FUNCTION_BLOCK FB_LUTDevice EXTENDS FD_Device 
VAR_INPUT
END_VAR

VAR_OUTPUT
END_VAR

VAR
	//===================== Variable
	eLTUPosition					: E_LTUPosition;
	bCarrierPresent				: BOOL;
	bLTUFree							: BOOL;
	
	bReserved							: BOOL;
	eReservedBy						: E_Convoyer;
	
	
	
	//===================== Instance
	fbPneuCyl3Pos_AxisZ								: FB_PneuCyl_3Pos     	 (GVL_Customer.C_Name_LTUPneuClyZ,
																															GVL_Customer.C_ID_LTUPneuClyZ
																										  				); 
																													
	fbStopperLut											: FB_PneuCyl_Stopper     (GVL_Customer.C_Name_LUTStopper,
																															GVL_Customer.C_ID_LUTStopper
																										  			 );																												
																													
	fbLUTLightBarrier									: FB_Input					  		(GVL_Customer.C_Name_LUTLightBarrier,
																															GVL_Customer.C_ID_LUTLightBarrier
																										  				);																																										
	
	fbLUTSimpleMotor									: FB_SimpleMotor      		(GVL_Customer.C_Name_LUTDcMotor,
																															GVL_Customer.C_ID_LUTSimpleMotor
																										  				);

																										
END_VAR

VAR CONSTANT
	// --------------------------Base------------------
	C_SeqStep_OnBasePos_Start								: UINT :=  20; 
	C_SeqStep_OnBasePos_WaitOpMode					: UINT :=  30;
	C_SeqStep_OnBasePos_Done								: UINT :=  100; 
	
	// --------------------------Auto Sequence------------------
	
	C_SeqStep_Auto_Start										: UINT :=  200;
	C_SeqStep_Auto_End											: UINT :=  400;
END_VAR


//******* Important and necessary
SUPER^();  
//====================================
IF NOT Enable THEN RETURN; END_IF

fbPneuCyl3Pos_AxisZ();
fbStopperLut();
fbLUTLightBarrier();
fbLUTSimpleMotor();

PROPERTY CarrierPresent : BOOL
GET
CarrierPresent := bCarrierPresent;
END_GET
SET
bCarrierPresent := CarrierPresent;
END_SET
END_PROPERTY

//FB_Init ist immer implizit verfügbar und wird primär für die Initialisierung verwendet.
//Der Rückgabewert wird nicht ausgewertet. Für gezielte Einflussnahme können Sie
//die Methoden explizit deklarieren und darin mit dem Standard-Initialisierungscode 
//zusätzlichen Code bereitstellen. Sie können den Rückgabewert auswerten.
METHOD FB_Init: BOOL
VAR_INPUT    
	bInitRetains					: BOOL; 					// TRUE: Die Retain-Variablen werden initialisiert (Reset warm / Reset kalt)    
	bInCopyCode						: BOOL;  					// TRUE: Die Instanz wird danach in den Kopiercode kopiert (Online-Change)
	
	I_Name                : STRING;         //  Name
	I_ID                  : UINT;           // ID
  I_itfOwner					  : ITF_Owner;      // owner 
END_VAR
END_METHOD

PROPERTY LTUFree : BOOL
GET

LTUFree := bLTUFree;
END_GET
SET
bLTUFree := LTUFree;
END_SET
END_PROPERTY

PROPERTY LTUPosition : E_LTUPosition
GET
LTUPosition := eLTUPosition;
END_GET
SET
eLTUPosition := LTUPosition;
END_SET
END_PROPERTY

METHOD mAutomatic : E_CmdState
VAR_INPUT
	I_bExecute	: BOOL;
END_VAR
END_METHOD

METHOD mCmdExec_Auto : E_CmdState
VAR_INPUT
END_VAR

CASE SequenceID OF

  //******************************************************* Idle 
  C_SeqStep_Idle: 
  	SequenceID       :=  C_SeqStep_Start;
  
  //****************************************************** Start
  C_SeqStep_Start:
  	
  	SequenceID       :=  C_SeqStep_OnBasePos_Start;
	C_SeqStep_OnBasePos_Start:
	
		SequenceID       :=  C_SeqStep_Done;;
	
//	C_SeqStep_OnBasePos_Start:
	
	
//	C_SeqStep_OnBasePos_Start:
	
	
  C_SeqStep_Error: 
    //************* all FB reset

		//************* 
    mCmdExec_Auto := mDone(); 
  //**********************Done 
  	
 	C_SeqStep_Done:
  	mCmdExec_Auto := mDone();

END_CASE
END_METHOD

METHOD mCmdExec_Homing : E_CmdState
VAR_INPUT
END_VAR

CASE SequenceID OF

  //******************************************************* Idle 
  C_SeqStep_Idle: 
  	SequenceID       :=  C_SeqStep_Start;
  
  //****************************************************** Start
  C_SeqStep_Start:
   
  	SequenceID       :=  C_SeqStep_Done;
	
  C_SeqStep_Error: 
    //************* all FB reset

		//************* 
    mCmdExec_Homing := mDone(); 
  //**********************Done 
 
 	C_SeqStep_Done:
  	mCmdExec_Homing := mDone();

END_CASE
END_METHOD

METHOD mCmdExec_MoveBottom : E_CmdState
VAR_INPUT
	I_bExecute					: BOOL;
END_VAR

VAR
	L_eCmdState 					: E_CmdState;
END_VAR
// No command requested.
IF NOT I_bExecute 
	THEN
  	mCmdExec_MoveMiddle := E_CmdState.Idle;
    RETURN;
END_IF

// Move vertical axis to TOP.
L_eCmdState := fbPneuCyl3Pos_AxisZ.mCallBottom(TRUE);
CASE L_eCmdState OF
	E_CmdState.Succeeded:
  	mCmdExec_MoveBottom := E_CmdState.Succeeded;
  E_CmdState.Busy:
  	mCmdExec_MoveBottom := E_CmdState.Busy;
ELSE
	mCmdExec_MoveBottom := L_eCmdState;
END_CASE
END_METHOD

METHOD mCmdExec_MoveMiddle : E_CmdState
VAR_INPUT
	I_bExecute					: BOOL;
END_VAR

VAR
	L_eCmdState 					: E_CmdState;
END_VAR
// No command requested.
IF NOT I_bExecute 
	THEN
  	mCmdExec_MoveMiddle := E_CmdState.Idle;
    RETURN;
END_IF

// Move vertical axis to TOP.
L_eCmdState := fbPneuCyl3Pos_AxisZ.mCallMiddle(TRUE);
CASE L_eCmdState OF
	E_CmdState.Succeeded:
  	mCmdExec_MoveMiddle := E_CmdState.Succeeded;
  E_CmdState.Busy:
  	mCmdExec_MoveMiddle := E_CmdState.Busy;
ELSE
	mCmdExec_MoveMiddle := L_eCmdState;
END_CASE
END_METHOD

METHOD mCmdExec_MoveTop : E_CmdState
VAR_INPUT
	I_bExecute					: BOOL;
END_VAR

VAR
	L_eCmdState 					: E_CmdState;
END_VAR
// No command requested.
IF NOT I_bExecute 
	THEN
  	mCmdExec_MoveTop := E_CmdState.Idle;
    RETURN;
END_IF

// Move vertical axis to TOP.
L_eCmdState := fbPneuCyl3Pos_AxisZ.mCallTop(TRUE);
CASE L_eCmdState OF
	E_CmdState.Succeeded:
  	mCmdExec_MoveTop := E_CmdState.Succeeded;
  E_CmdState.Busy:
  	mCmdExec_MoveTop := E_CmdState.Busy;
ELSE
	mCmdExec_MoveTop := L_eCmdState;
END_CASE
END_METHOD

METHOD mCmdExec_Service : E_CmdState
VAR_INPUT
END_VAR
;
END_METHOD

METHOD mCmdExec_TransferTop : E_CmdState
VAR_INPUT
	I_bExecute					: BOOL;
END_VAR
// No command requested.
IF NOT I_bExecute THEN
    fbLUTSimpleMotor.mStopMotor(TRUE);
    mCmdExec_TransferTop := E_CmdState.Idle;
    RETURN;
END_IF

// Start LTU motor for top transfer.
fbLUTSimpleMotor.mStartMotor(TRUE);

// Wait  carrier leaves LTU.
IF NOT fbStopperLut.CarriePresent 
	THEN
    fbLUTSimpleMotor.mStopMotor(TRUE);
    mCmdExec_TransferTop := E_CmdState.Succeeded;
    RETURN;
END_IF

mCmdExec_TransferTop := E_CmdState.Busy;
END_METHOD

METHOD mHold : E_CmdState
VAR_INPUT
	I_bExecute	: BOOL;
END_VAR

SUPER^.mHold(I_bExecute);
END_METHOD

METHOD mHome : E_CmdState
VAR_INPUT
	I_bExecute	: BOOL;
END_VAR

SUPER^.mHome(I_bExecute);
END_METHOD

METHOD mRelease : E_CmdState
VAR_INPUT
	I_bExecute	: BOOL;
END_VAR

SUPER^.mRelease(I_bExecute);
END_METHOD

METHOD mSequence : E_CmdState
VAR_INPUT
	I_bExecute				: BOOL;
END_VAR

VAR
	L_eState 					: E_CmdState;
END_VAR
mSequence := SUPER^.mSequence(I_bExecute);	


// Generic checks from parent
L_eState := SUPER^.mSequence(I_bExecute := I_bExecute);

IF L_eState <> E_CmdState.Busy 
	THEN
    mSequence := L_eState;
    RETURN;
END_IF

CASE Mode OF
	E_Mode.Homing:
		mSequence := mCmdExec_Homing();
		
	E_Mode.Auto:
		mSequence := mCmdExec_Auto();
		
	E_Mode.Service:
		mSequence := mCmdExec_Service();
		
END_CASE
END_METHOD

METHOD mService : E_CmdState
VAR_INPUT
	I_bExecute	: BOOL;
END_VAR

SUPER^.mService(I_bExecute);
END_METHOD

METHOD mStop : E_CmdState
VAR_INPUT
	I_bExecute	: BOOL;
END_VAR

SUPER^.mStop(I_bExecute);
END_METHOD

PROPERTY ReservedBy : E_Convoyer
GET
ReservedBy := eReservedBy;
END_GET
SET
eReservedBy := ReservedBy;
END_SET
END_PROPERTY

END_FUNCTION_BLOCK

(* stored: Version 1.1.0.1, ProductVersion 3.1.4026.18
   POU FB_LUTDevice: Id {1d37f6f4-ced3-4fc7-b8fb-537fe5b0ee0b}, SpecialFunc None
   Folder 01 Properties: Id {01153c84-2cbf-4774-9afe-06465af82a17}
   Folder 02 Methodes: Id {1154e57b-5607-4e8c-9894-d39905ffa9c5}
   Folder 100 CmdExecute: Id {737ecdee-bdd3-4011-be43-9c8053143eb0}
   Property CarrierPresent: Id {b074603b-40b1-4657-ab62-b1cd6acb861f}
   Get Get: Id {88207567-04e5-4568-82f0-781cf9a61ad4}
   Set Set: Id {fd122f58-f442-4621-8637-9e667fca0acd}
   Method FB_Init: Id {4e8aa732-d3ac-4d90-bbea-84986dfc142d}
   Property LTUFree: Id {1f84a690-a1f2-456d-ad2b-bc5117437904}
   Get Get: Id {d00d9a6b-7aca-4015-aa9d-f54e3711617d}
   Set Set: Id {d538fb44-3dfc-4c3c-8b31-3a15c25ffd6c}
   Property LTUPosition: Id {c1f15a68-48c8-460e-be2e-811c99b99676}
   Get Get: Id {6ea8e49b-49a8-4199-a325-4e224d8d6684}
   Set Set: Id {a1718f28-a922-45a4-926f-c3a142e1f8ee}
   Method mAutomatic: Id {1a363c95-a5ab-493c-a24f-fc972dc90c4d}
   Method mCmdExec_Auto: Id {90a7dbfb-cbde-4eb5-878d-9d7c2e891557}
   Method mCmdExec_Homing: Id {ec212c1f-d213-4550-add5-c0351f9927e9}
   Method mCmdExec_MoveBottom: Id {8febe5ee-97da-4ab2-9486-5866194a4d14}
   Method mCmdExec_MoveMiddle: Id {31257785-c557-43e8-9c51-32cde10873f6}
   Method mCmdExec_MoveTop: Id {4ff0852f-f39d-4fd3-895f-9db63096116e}
   Method mCmdExec_Service: Id {b17d27f6-62e0-420a-b1d7-d447cfe9cb9d}
   Method mCmdExec_TransferTop: Id {d2f6dd01-c2ed-4343-891b-6738e835be35}
   Method mHold: Id {9c6da647-9b3a-4008-822a-f46989735258}
   Method mHome: Id {49ad83dc-2a17-49c4-8611-ff23b94da67e}
   Method mRelease: Id {371d93b7-c4a5-4cdb-81ce-2ec14cd8d7cb}
   Method mSequence: Id {34a06eeb-9098-4b67-9089-0adc32ada112}
   Method mService: Id {6e836c74-9634-4f57-9fa1-a7cf3b465050}
   Method mStop: Id {d84c7b32-8c21-42a5-9b35-6c7a9a260b8f}
   Property ReservedBy: Id {cb2eae19-49dd-472f-ae1a-bd6a0377a00b}
   Get Get: Id {794b05e1-e352-4d18-bf73-38d2b088bb67}
   Set Set: Id {7ecf7796-1c1a-4216-9263-351ab44afc8c} *)
